//     Term 163 (AT2000-0250)/CC Inputs/Current actual value Ch.6 <-> Data Pointer/CurrentActualValues[5]
//     Term 163 (AT2000-0250)/CC Inputs/Current actual value Ch.7 <-> Data Pointer/CurrentActualValues[6]
//     Term 163 (AT2000-0250)/CC Inputs/Current actual value Ch.8 <-> Data Pointer/CurrentActualValues[7]
//     Term 163 (AT2000-0250)/CC Inputs/Current actual value Ch.9 <-> Data Pointer/CurrentActualValues[8]
//     Term 163 (AT2000-0250)/CC Inputs/Status <-> Data Pointer/Status
//     Term 163 (AT2000-0250)/CC Outputs/Control <-> Data Pointer/Control
//     Term 163 (AT2000-0250)/CC Outputs/Current setpoint value Ch.1 <-> Data Pointer/CurrentSetpointValues[0]
//     Term 163 (AT2000-0250)/CC Outputs/Current setpoint value Ch.10 <-> Data Pointer/CurrentSetpointValues[9]
//     Term 163 (AT2000-0250)/CC Outputs/Current setpoint value Ch.11 <-> Data Pointer/CurrentSetpointValues[10]
//     Term 163 (AT2000-0250)/CC Outputs/Current setpoint value Ch.12 <-> Data Pointer/CurrentSetpointValues[11]
//     Term 163 (AT2000-0250)/CC Outputs/Current setpoint value Ch.13 <-> Data Pointer/CurrentSetpointValues[12]
//     Term 163 (AT2000-0250)/CC Outputs/Current setpoint value Ch.14 <-> Data Pointer/CurrentSetpointValues[13]
//     Term 163 (AT2000-0250)/CC Outputs/Current setpoint value Ch.15 <-> Data Pointer/CurrentSetpointValues[14]
//     Term 163 (AT2000-0250)/CC Outputs/Current setpoint value Ch.2 <-> Data Pointer/CurrentSetpointValues[1]
//     Term 163 (AT2000-0250)/CC Outputs/Current setpoint value Ch.3 <-> Data Pointer/CurrentSetpointValues[2]
//     Term 163 (AT2000-0250)/CC Outputs/Current setpoint value Ch.4 <-> Data Pointer/CurrentSetpointValues[3]
//     Term 163 (AT2000-0250)/CC Outputs/Current setpoint value Ch.5 <-> Data Pointer/CurrentSetpointValues[4]
//     Term 163 (AT2000-0250)/CC Outputs/Current setpoint value Ch.6 <-> Data Pointer/CurrentSetpointValues[5]
//     Term 163 (AT2000-0250)/CC Outputs/Current setpoint value Ch.7 <-> Data Pointer/CurrentSetpointValues[6]
//     Term 163 (AT2000-0250)/CC Outputs/Current setpoint value Ch.8 <-> Data Pointer/CurrentSetpointValues[7]
//     Term 163 (AT2000-0250)/CC Outputs/Current setpoint value Ch.9 <-> Data Pointer/CurrentSetpointValues[8]
//     Term 163 (AT2000-0250)/Term 164 (AT2000-5250)/FB Inputs/Value Channel 01 <-> Data Pointer/RawPositionValues[0]
//     Term 163 (AT2000-0250)/Term 164 (AT2000-5250)/FB Inputs/Value Channel 02 <-> Data Pointer/RawPositionValues[1]
//     Term 163 (AT2000-0250)/Term 164 (AT2000-5250)/FB Inputs/Value Channel 03 <-> Data Pointer/RawPositionValues[2]
//     Term 163 (AT2000-0250)/Term 164 (AT2000-5250)/FB Inputs/Value Channel 04 <-> Data Pointer/RawPositionValues[3]
//     Term 163 (AT2000-0250)/Term 164 (AT2000-5250)/FB Inputs/Value Channel 05 <-> Data Pointer/RawPositionValues[4]
//     Term 163 (AT2000-0250)/Term 164 (AT2000-5250)/FB Inputs/Value Channel 06 <-> Data Pointer/RawPositionValues[5]
//     Term 163 (AT2000-0250)/Term 164 (AT2000-5250)/FB Inputs/Value Channel 07 <-> Data Pointer/RawPositionValues[6]
//     Term 163 (AT2000-0250)/Term 164 (AT2000-5250)/FB Inputs/Value Channel 08 <-> Data Pointer/RawPositionValues[7]
//     Term 163 (AT2000-0250)/Term 164 (AT2000-5250)/FB Inputs/Value Channel 09 <-> Data Pointer/RawPositionValues[8]
//     Term 163 (AT2000-0250)/Term 164 (AT2000-5250)/FB Inputs/Value Channel 10 <-> Data Pointer/RawPositionValues[9]
//     Term 163 (AT2000-0250)/Term 164 (AT2000-5250)/FB Inputs/Value Channel 11 <-> Data Pointer/RawPositionValues[10]
//     Term 163 (AT2000-0250)/Term 164 (AT2000-5250)/FB Inputs/Value Channel 12 <-> Data Pointer/RawPositionValues[11]
//     Term 163 (AT2000-0250)/Term 164 (AT2000-5250)/FB Inputs/Value Channel 13 <-> Data Pointer/RawPositionValues[12]
//     Term 163 (AT2000-0250)/Term 164 (AT2000-5250)/FB Inputs/Value Channel 14 <-> Data Pointer/RawPositionValues[13]
//     Term 163 (AT2000-0250)/Term 164 (AT2000-5250)/FB Inputs/Value Channel 15 <-> Data Pointer/RawPositionValues[14]
//     Term 163 (AT2000-0250)/Term 164 (AT2000-5250)/FB Inputs/Value Channel 16 <-> Data Pointer/RawPositionValues[15]
//     Term 163 (AT2000-0250)/Term 164 (AT2000-5250)/FB Inputs/Value Channel 17 <-> Data Pointer/RawPositionValues[16]
//     Term 163 (AT2000-0250)/Term 164 (AT2000-5250)/FB Inputs/Value Channel 18 <-> Data Pointer/RawPositionValues[17]
//     Term 163 (AT2000-0250)/Term 164 (AT2000-5250)/FB Inputs/Value Channel 19 <-> Data Pointer/RawPositionValues[18]
//     Term 163 (AT2000-0250)/Term 164 (AT2000-5250)/FB Inputs/Value Channel 20 <-> Data Pointer/RawPositionValues[19]
//     Term 163 (AT2000-0250)/Term 164 (AT2000-5250)/FB Inputs/Value Channel 21 <-> Data Pointer/RawPositionValues[20]
//     Term 163 (AT2000-0250)/Term 164 (AT2000-5250)/FB Inputs/Value Channel 22 <-> Data Pointer/RawPositionValues[21]
//     Term 163 (AT2000-0250)/Term 164 (AT2000-5250)/FB Inputs/Value Channel 23 <-> Data Pointer/RawPositionValues[22]
//     Term 163 (AT2000-0250)/Term 164 (AT2000-5250)/FB Inputs/Value Channel 24 <-> Data Pointer/RawPositionValues[23]
//     Term 163 (AT2000-0250)/Term 164 (AT2000-5250)/FB Inputs/Value Channel 25 <-> Data Pointer/RawPositionValues[24]
//     Term 163 (AT2000-0250)/Term 164 (AT2000-5250)/FB Inputs/Value Channel 26 <-> Data Pointer/RawPositionValues[25]
//     Term 163 (AT2000-0250)/Term 164 (AT2000-5250)/FB Inputs/Value Channel 27 <-> Data Pointer/RawPositionValues[26]
//     Term 163 (AT2000-0250)/Term 164 (AT2000-5250)/FB Inputs/Value Channel 28 <-> Data Pointer/RawPositionValues[27]
//     Term 163 (AT2000-0250)/Term 164 (AT2000-5250)/FB Inputs/Value Channel 29 <-> Data Pointer/RawPositionValues[28]
//     Term 163 (AT2000-0250)/Term 164 (AT2000-5250)/FB Inputs/Value Channel 30 <-> Data Pointer/RawPositionValues[29]
//     Term 163 (AT2000-0250)/Term 164 (AT2000-5250)/FB Inputs/Value Channel 31 <-> Data Pointer/RawPositionValues[30]
//     Term 163 (AT2000-0250)/Term 164 (AT2000-5250)/FB Inputs/Value Channel 32 <-> Data Pointer/RawPositionValues[31]
//   (this object) <-> TcCOM Objects/XtsProcessingUnit 1/Part 1/Module 83
//     Term 165 (AT2050-0500)/CC Inputs/Current actual value Ch.1 <-> Data Pointer/CurrentActualValues[0]
//     Term 165 (AT2050-0500)/CC Inputs/Current actual value Ch.10 <-> Data Pointer/CurrentActualValues[9]
//     Term 165 (AT2050-0500)/CC Inputs/Current actual value Ch.11 <-> Data Pointer/CurrentActualValues[10]
//     Term 165 (AT2050-0500)/CC Inputs/Current actual value Ch.12 <-> Data Pointer/CurrentActualValues[11]
//     Term 165 (AT2050-0500)/CC Inputs/Current actual value Ch.13 <-> Data Pointer/CurrentActualValues[12]
//     Term 165 (AT2050-0500)/CC Inputs/Current actual value Ch.14 <-> Data Pointer/CurrentActualValues[13]
//     Term 165 (AT2050-0500)/CC Inputs/Current actual value Ch.15 <-> Data Pointer/CurrentActualValues[14]
//     Term 165 (AT2050-0500)/CC Inputs/Current actual value Ch.2 <-> Data Pointer/CurrentActualValues[1]
//     Term 165 (AT2050-0500)/CC Inputs/Current actual value Ch.3 <-> Data Pointer/CurrentActualValues[2]
//     Term 165 (AT2050-0500)/CC Inputs/Current actual value Ch.4 <-> Data Pointer/CurrentActualValues[3]
//     Term 165 (AT2050-0500)/CC Inputs/Current actual value Ch.5 <-> Data Pointer/CurrentActualValues[4]
//     Term 165 (AT2050-0500)/CC Inputs/Current actual value Ch.6 <-> Data Pointer/CurrentActualValues[5]
//     Term 165 (AT2050-0500)/CC Inputs/Current actual value Ch.7 <-> Data Pointer/CurrentActualValues[6]
//     Term 165 (AT2050-0500)/CC Inputs/Current actual value Ch.8 <-> Data Pointer/CurrentActualValues[7]
//     Term 165 (AT2050-0500)/CC Inputs/Current actual value Ch.9 <-> Data Pointer/CurrentActualValues[8]
//     Term 165 (AT2050-0500)/CC Inputs/Status <-> Data Pointer/Status
//     Term 165 (AT2050-0500)/CC Outputs/Control <-> Data Pointer/Control
//     Term 165 (AT2050-0500)/CC Outputs/Current setpoint value Ch.1 <-> Data Pointer/CurrentSetpointValues[0]
//     Term 165 (AT2050-0500)/CC Outputs/Current setpoint value Ch.10 <-> Data Pointer/CurrentSetpointValues[9]
//     Term 165 (AT2050-0500)/CC Outputs/Current setpoint value Ch.11 <-> Data Pointer/CurrentSetpointValues[10]
//     Term 165 (AT2050-0500)/CC Outputs/Current setpoint value Ch.12 <-> Data Pointer/CurrentSetpointValues[11]
//     Term 165 (AT2050-0500)/CC Outputs/Current setpoint value Ch.13 <-> Data Pointer/CurrentSetpointValues[12]
//     Term 165 (AT2050-0500)/CC Outputs/Current setpoint value Ch.14 <-> Data Pointer/CurrentSetpointValues[13]
//     Term 165 (AT2050-0500)/CC Outputs/Current setpoint value Ch.15 <-> Data Pointer/CurrentSetpointValues[14]
//     Term 165 (AT2050-0500)/CC Outputs/Current setpoint value Ch.2 <-> Data Pointer/CurrentSetpointValues[1]
//     Term 165 (AT2050-0500)/CC Outputs/Current setpoint value Ch.3 <-> Data Pointer/CurrentSetpointValues[2]
//     Term 165 (AT2050-0500)/CC Outputs/Current setpoint value Ch.4 <-> Data Pointer/CurrentSetpointValues[3]
//     Term 165 (AT2050-0500)/CC Outputs/Current setpoint value Ch.5 <-> Data Pointer/CurrentSetpointValues[4]
//     Term 165 (AT2050-0500)/CC Outputs/Current setpoint value Ch.6 <-> Data Pointer/CurrentSetpointValues[5]
//     Term 165 (AT2050-0500)/CC Outputs/Current setpoint value Ch.7 <-> Data Pointer/CurrentSetpointValues[6]
//     Term 165 (AT2050-0500)/CC Outputs/Current setpoint value Ch.8 <-> Data Pointer/CurrentSetpointValues[7]
//     Term 165 (AT2050-0500)/CC Outputs/Current setpoint value Ch.9 <-> Data Pointer/CurrentSetpointValues[8]
//     Term 165 (AT2050-0500)/Term 166 (AT2050-5500)/FB Inputs/Value Channel 01 <-> Data Pointer/RawPositionValues[0]
//     Term 165 (AT2050-0500)/Term 166 (AT2050-5500)/FB Inputs/Value Channel 02 <-> Data Pointer/RawPositionValues[1]
//     Term 165 (AT2050-0500)/Term 166 (AT2050-5500)/FB Inputs/Value Channel 03 <-> Data Pointer/RawPositionValues[2]
//     Term 165 (AT2050-0500)/Term 166 (AT2050-5500)/FB Inputs/Value Channel 04 <-> Data Pointer/RawPositionValues[3]
//     Term 165 (AT2050-0500)/Term 166 (AT2050-5500)/FB Inputs/Value Channel 05 <-> Data Pointer/RawPositionValues[4]
//     Term 165 (AT2050-0500)/Term 166 (AT2050-5500)/FB Inputs/Value Channel 06 <-> Data Pointer/RawPositionValues[5]
//     Term 165 (AT2050-0500)/Term 166 (AT2050-5500)/FB Inputs/Value Channel 07 <-> Data Pointer/RawPositionValues[6]
//     Term 165 (AT2050-0500)/Term 166 (AT2050-5500)/FB Inputs/Value Channel 08 <-> Data Pointer/RawPositionValues[7]
//     Term 165 (AT2050-0500)/Term 166 (AT2050-5500)/FB Inputs/Value Channel 09 <-> Data Pointer/RawPositionValues[8]
//     Term 165 (AT2050-0500)/Term 166 (AT2050-5500)/FB Inputs/Value Channel 10 <-> Data Pointer/RawPositionValues[9]
//     Term 165 (AT2050-0500)/Term 166 (AT2050-5500)/FB Inputs/Value Channel 11 <-> Data Pointer/RawPositionValues[10]
//     Term 165 (AT2050-0500)/Term 166 (AT2050-5500)/FB Inputs/Value Channel 12 <-> Data Pointer/RawPositionValues[11]
//     Term 165 (AT2050-0500)/Term 166 (AT2050-5500)/FB Inputs/Value Channel 13 <-> Data Pointer/RawPositionValues[12]
//     Term 165 (AT2050-0500)/Term 166 (AT2050-5500)/FB Inputs/Value Channel 14 <-> Data Pointer/RawPositionValues[13]
//     Term 165 (AT2050-0500)/Term 166 (AT2050-5500)/FB Inputs/Value Channel 15 <-> Data Pointer/RawPositionValues[14]
//     Term 165 (AT2050-0500)/Term 166 (AT2050-5500)/FB Inputs/Value Channel 16 <-> Data Pointer/RawPositionValues[15]
//     Term 165 (AT2050-0500)/Term 166 (AT2050-5500)/FB Inputs/Value Channel 17 <-> Data Pointer/RawPositionValues[16]
//     Term 165 (AT2050-0500)/Term 166 (AT2050-5500)/FB Inputs/Value Channel 18 <-> Data Pointer/RawPositionValues[17]
//     Term 165 (AT2050-0500)/Term 166 (AT2050-5500)/FB Inputs/Value Channel 19 <-> Data Pointer/RawPositionValues[18]
//     Term 165 (AT2050-0500)/Term 166 (AT2050-5500)/FB Inputs/Value Channel 20 <-> Data Pointer/RawPositionValues[19]
//     Term 165 (AT2050-0500)/Term 166 (AT2050-5500)/FB Inputs/Value Channel 21 <-> Data Pointer/RawPositionValues[20]
//     Term 165 (AT2050-0500)/Term 166 (AT2050-5500)/FB Inputs/Value Channel 22 <-> Data Pointer/RawPositionValues[21]
//     Term 165 (AT2050-0500)/Term 166 (AT2050-5500)/FB Inputs/Value Channel 23 <-> Data Pointer/RawPositionValues[22]
//     Term 165 (AT2050-0500)/Term 166 (AT2050-5500)/FB Inputs/Value Channel 24 <-> Data Pointer/RawPositionValues[23]
//     Term 165 (AT2050-0500)/Term 166 (AT2050-5500)/FB Inputs/Value Channel 25 <-> Data Pointer/RawPositionValues[24]
//     Term 165 (AT2050-0500)/Term 166 (AT2050-5500)/FB Inputs/Value Channel 26 <-> Data Pointer/RawPositionValues[25]
//     Term 165 (AT2050-0500)/Term 166 (AT2050-5500)/FB Inputs/Value Channel 27 <-> Data Pointer/RawPositionValues[26]
//     Term 165 (AT2050-0500)/Term 166 (AT2050-5500)/FB Inputs/Value Channel 28 <-> Data Pointer/RawPositionValues[27]
//     Term 165 (AT2050-0500)/Term 166 (AT2050-5500)/FB Inputs/Value Channel 29 <-> Data Pointer/RawPositionValues[28]
//     Term 165 (AT2050-0500)/Term 166 (AT2050-5500)/FB Inputs/Value Channel 30 <-> Data Pointer/RawPositionValues[29]
//     Term 165 (AT2050-0500)/Term 166 (AT2050-5500)/FB Inputs/Value Channel 31 <-> Data Pointer/RawPositionValues[30]
//     Term 165 (AT2050-0500)/Term 166 (AT2050-5500)/FB Inputs/Value Channel 32 <-> Data Pointer/RawPositionValues[31]
//   (this object) <-> TcCOM Objects/XtsProcessingUnit 1/Part 1/Module 84
//     Term 167 (AT2050-0501)/CC Inputs/Current actual value Ch.1 <-> Data Pointer/CurrentActualValues[0]
//     Term 167 (AT2050-0501)/CC Inputs/Current actual value Ch.10 <-> Data Pointer/CurrentActualValues[9]
//     Term 167 (AT2050-0501)/CC Inputs/Current actual value Ch.11 <-> Data Pointer/CurrentActualValues[10]
//     Term 167 (AT2050-0501)/CC Inputs/Current actual value Ch.12 <-> Data Pointer/CurrentActualValues[11]
//     Term 167 (AT2050-0501)/CC Inputs/Current actual value Ch.13 <-> Data Pointer/CurrentActualValues[12]
//     Term 167 (AT2050-0501)/CC Inputs/Current actual value Ch.14 <-> Data Pointer/CurrentActualValues[13]
//     Term 167 (AT2050-0501)/CC Inputs/Current actual value Ch.15 <-> Data Pointer/CurrentActualValues[14]
//     Term 167 (AT2050-0501)/CC Inputs/Current actual value Ch.2 <-> Data Pointer/CurrentActualValues[1]
//     Term 167 (AT2050-0501)/CC Inputs/Current actual value Ch.3 <-> Data Pointer/CurrentActualValues[2]
//     Term 167 (AT2050-0501)/CC Inputs/Current actual value Ch.4 <-> Data Pointer/CurrentActualValues[3]
//     Term 167 (AT2050-0501)/CC Inputs/Current actual value Ch.5 <-> Data Pointer/CurrentActualValues[4]
//     Term 167 (AT2050-0501)/CC Inputs/Current actual value Ch.6 <-> Data Pointer/CurrentActualValues[5]
//     Term 167 (AT2050-0501)/CC Inputs/Current actual value Ch.7 <-> Data Pointer/CurrentActualValues[6]
//     Term 167 (AT2050-0501)/CC Inputs/Current actual value Ch.8 <-> Data Pointer/CurrentActualValues[7]
//     Term 167 (AT2050-0501)/CC Inputs/Current actual value Ch.9 <-> Data Pointer/CurrentActualValues[8]
//     Term 167 (AT2050-0501)/CC Inputs/Status <-> Data Pointer/Status
//     Term 167 (AT2050-0501)/CC Outputs/Control <-> Data Pointer/Control
//     Term 167 (AT2050-0501)/CC Outputs/Current setpoint value Ch.1 <-> Data Pointer/CurrentSetpointValues[0]
//     Term 167 (AT2050-0501)/CC Outputs/Current setpoint value Ch.10 <-> Data Pointer/CurrentSetpointValues[9]
//     Term 167 (AT2050-0501)/CC Outputs/Current setpoint value Ch.11 <-> Data Pointer/CurrentSetpointValues[10]
//     Term 167 (AT2050-0501)/CC Outputs/Current setpoint value Ch.12 <-> Data Pointer/CurrentSetpointValues[11]
//     Term 167 (AT2050-0501)/CC Outputs/Current setpoint value Ch.13 <-> Data Pointer/CurrentSetpointValues[12]
//     Term 167 (AT2050-0501)/CC Outputs/Current setpoint value Ch.14 <-> Data Pointer/CurrentSetpointValues[13]
//     Term 167 (AT2050-0501)/CC Outputs/Current setpoint value Ch.15 <-> Data Pointer/CurrentSetpointValues[14]
//     Term 167 (AT2050-0501)/CC Outputs/Current setpoint value Ch.2 <-> Data Pointer/CurrentSetpointValues[1]
//     Term 167 (AT2050-0501)/CC Outputs/Current setpoint value Ch.3 <-> Data Pointer/CurrentSetpointValues[2]
//     Term 167 (AT2050-0501)/CC Outputs/Current setpoint value Ch.4 <-> Data Pointer/CurrentSetpointValues[3]
//     Term 167 (AT2050-0501)/CC Outputs/Current setpoint value Ch.5 <-> Data Pointer/CurrentSetpointValues[4]
//     Term 167 (AT2050-0501)/CC Outputs/Current setpoint value Ch.6 <-> Data Pointer/CurrentSetpointValues[5]
//     Term 167 (AT2050-0501)/CC Outputs/Current setpoint value Ch.7 <-> Data Pointer/CurrentSetpointValues[6]
//     Term 167 (AT2050-0501)/CC Outputs/Current setpoint value Ch.8 <-> Data Pointer/CurrentSetpointValues[7]
//     Term 167 (AT2050-0501)/CC Outputs/Current setpoint value Ch.9 <-> Data Pointer/CurrentSetpointValues[8]
//     Term 167 (AT2050-0501)/Term 168 (AT2050-5501)/FB Inputs/Value Channel 01 <-> Data Pointer/RawPositionValues[0]
//     Term 167 (AT2050-0501)/Term 168 (AT2050-5501)/FB Inputs/Value Channel 02 <-> Data Pointer/RawPositionValues[1]
//     Term 167 (AT2050-0501)/Term 168 (AT2050-5501)/FB Inputs/Value Channel 03 <-> Data Pointer/RawPositionValues[2]
//     Term 167 (AT2050-0501)/Term 168 (AT2050-5501)/FB Inputs/Value Channel 04 <-> Data Pointer/RawPositionValues[3]
//     Term 167 (AT2050-0501)/Term 168 (AT2050-5501)/FB Inputs/Value Channel 05 <-> Data Pointer/RawPositionValues[4]
//     Term 167 (AT2050-0501)/Term 168 (AT2050-5501)/FB Inputs/Value Channel 06 <-> Data Pointer/RawPositionValues[5]
//     Term 167 (AT2050-0501)/Term 168 (AT2050-5501)/FB Inputs/Value Channel 07 <-> Data Pointer/RawPositionValues[6]
//     Term 167 (AT2050-0501)/Term 168 (AT2050-5501)/FB Inputs/Value Channel 08 <-> Data Pointer/RawPositionValues[7]
//     Term 167 (AT2050-0501)/Term 168 (AT2050-5501)/FB Inputs/Value Channel 09 <-> Data Pointer/RawPositionValues[8]
//     Term 167 (AT2050-0501)/Term 168 (AT2050-5501)/FB Inputs/Value Channel 10 <-> Data Pointer/RawPositionValues[9]
//     Term 167 (AT2050-0501)/Term 168 (AT2050-5501)/FB Inputs/Value Channel 11 <-> Data Pointer/RawPositionValues[10]
//     Term 167 (AT2050-0501)/Term 168 (AT2050-5501)/FB Inputs/Value Channel 12 <-> Data Pointer/RawPositionValues[11]
//     Term 167 (AT2050-0501)/Term 168 (AT2050-5501)/FB Inputs/Value Channel 13 <-> Data Pointer/RawPositionValues[12]
//     Term 167 (AT2050-0501)/Term 168 (AT2050-5501)/FB Inputs/Value Channel 14 <-> Data Pointer/RawPositionValues[13]
//     Term 167 (AT2050-0501)/Term 168 (AT2050-5501)/FB Inputs/Value Channel 15 <-> Data Pointer/RawPositionValues[14]
//     Term 167 (AT2050-0501)/Term 168 (AT2050-5501)/FB Inputs/Value Channel 16 <-> Data Pointer/RawPositionValues[15]
//     Term 167 (AT2050-0501)/Term 168 (AT2050-5501)/FB Inputs/Value Channel 17 <-> Data Pointer/RawPositionValues[16]
//     Term 167 (AT2050-0501)/Term 168 (AT2050-5501)/FB Inputs/Value Channel 18 <-> Data Pointer/RawPositionValues[17]
//     Term 167 (AT2050-0501)/Term 168 (AT2050-5501)/FB Inputs/Value Channel 19 <-> Data Pointer/RawPositionValues[18]
//     Term 167 (AT2050-0501)/Term 168 (AT2050-5501)/FB Inputs/Value Channel 20 <-> Data Pointer/RawPositionValues[19]
//     Term 167 (AT2050-0501)/Term 168 (AT2050-5501)/FB Inputs/Value Channel 21 <-> Data Pointer/RawPositionValues[20]
//     Term 167 (AT2050-0501)/Term 168 (AT2050-5501)/FB Inputs/Value Channel 22 <-> Data Pointer/RawPositionValues[21]
//     Term 167 (AT2050-0501)/Term 168 (AT2050-5501)/FB Inputs/Value Channel 23 <-> Data Pointer/RawPositionValues[22]
//     Term 167 (AT2050-0501)/Term 168 (AT2050-5501)/FB Inputs/Value Channel 24 <-> Data Pointer/RawPositionValues[23]
//     Term 167 (AT2050-0501)/Term 168 (AT2050-5501)/FB Inputs/Value Channel 25 <-> Data Pointer/RawPositionValues[24]
//     Term 167 (AT2050-0501)/Term 168 (AT2050-5501)/FB Inputs/Value Channel 26 <-> Data Pointer/RawPositionValues[25]
//     Term 167 (AT2050-0501)/Term 168 (AT2050-5501)/FB Inputs/Value Channel 27 <-> Data Pointer/RawPositionValues[26]
//     Term 167 (AT2050-0501)/Term 168 (AT2050-5501)/FB Inputs/Value Channel 28 <-> Data Pointer/RawPositionValues[27]
//     Term 167 (AT2050-0501)/Term 168 (AT2050-5501)/FB Inputs/Value Channel 29 <-> Data Pointer/RawPositionValues[28]
//     Term 167 (AT2050-0501)/Term 168 (AT2050-5501)/FB Inputs/Value Channel 30 <-> Data Pointer/RawPositionValues[29]
//     Term 167 (AT2050-0501)/Term 168 (AT2050-5501)/FB Inputs/Value Channel 31 <-> Data Pointer/RawPositionValues[30]
//     Term 167 (AT2050-0501)/Term 168 (AT2050-5501)/FB Inputs/Value Channel 32 <-> Data Pointer/RawPositionValues[31]
//   PLC1 Instance <-> NC-Task SAF/Axes/Mover Axis 1
//     PlcTask Inputs/MAIN.aMovers[1].Axis.Axis.NcToPlc <-> Outputs/ToPlc
//     PlcTask Outputs/MAIN.aMovers[1].Axis.Axis.PlcToNc <-> Inputs/FromPlc
//   PLC1 Instance <-> NC-Task SAF/Axes/Mover Axis 10
//     PlcTask Inputs/MAIN.aMovers[10].Axis.Axis.NcToPlc <-> Outputs/ToPlc
//     PlcTask Outputs/MAIN.aMovers[10].Axis.Axis.PlcToNc <-> Inputs/FromPlc
//   PLC1 Instance <-> NC-Task SAF/Axes/Mover Axis 100
//     PlcTask Inputs/MAIN.aMovers[100].Axis.Axis.NcToPlc <-> Outputs/ToPlc
//     PlcTask Outputs/MAIN.aMovers[100].Axis.Axis.PlcToNc <-> Inputs/FromPlc
//   PLC1 Instance <-> NC-Task SAF/Axes/Mover Axis 11
//     PlcTask Inputs/MAIN.aMovers[11].Axis.Axis.NcToPlc <-> Outputs/ToPlc
//     PlcTask Outputs/MAIN.aMovers[11].Axis.Axis.PlcToNc <-> Inputs/FromPlc
//   PLC1 Instance <-> NC-Task SAF/Axes/Mover Axis 12
//     PlcTask Inputs/MAIN.aMovers[12].Axis.Axis.NcToPlc <-> Outputs/ToPlc
//     PlcTask Outputs/MAIN.aMovers[12].Axis.Axis.PlcToNc <-> Inputs/FromPlc
//   PLC1 Instance <-> NC-Task SAF/Axes/Mover Axis 13
//     PlcTask Inputs/MAIN.aMovers[13].Axis.Axis.NcToPlc <-> Outputs/ToPlc
//     PlcTask Outputs/MAIN.aMovers[13].Axis.Axis.PlcToNc <-> Inputs/FromPlc
//   PLC1 Instance <-> NC-Task SAF/Axes/Mover Axis 14
//     PlcTask Inputs/MAIN.aMovers[14].Axis.Axis.NcToPlc <-> Outputs/ToPlc
//     PlcTask Outputs/MAIN.aMovers[14].Axis.Axis.PlcToNc <-> Inputs/FromPlc
//   PLC1 Instance <-> NC-Task SAF/Axes/Mover Axis 15
//     PlcTask Inputs/MAIN.aMovers[15].Axis.Axis.NcToPlc <-> Outputs/ToPlc
//     PlcTask Outputs/MAIN.aMovers[15].Axis.Axis.PlcToNc <-> Inputs/FromPlc
//   PLC1 Instance <-> NC-Task SAF/Axes/Mover Axis 16
//     PlcTask Inputs/MAIN.aMovers[16].Axis.Axis.NcToPlc <-> Outputs/ToPlc
//     PlcTask Outputs/MAIN.aMovers[16].Axis.Axis.PlcToNc <-> Inputs/FromPlc
//   PLC1 Instance <-> NC-Task SAF/Axes/Mover Axis 17
//     PlcTask Inputs/MAIN.aMovers[17].Axis.Axis.NcToPlc <-> Outputs/ToPlc
//     PlcTask Outputs/MAIN.aMovers[17].Axis.Axis.PlcToNc <-> Inputs/FromPlc
//   PLC1 Instance <-> NC-Task SAF/Axes/Mover Axis 18
//     PlcTask Inputs/MAIN.aMovers[18].Axis.Axis.NcToPlc <-> Outputs/ToPlc
//     PlcTask Outputs/MAIN.aMovers[18].Axis.Axis.PlcToNc <-> Inputs/FromPlc
//   PLC1 Instance <-> NC-Task SAF/Axes/Mover Axis 19
//     PlcTask Inputs/MAIN.aMovers[19].Axis.Axis.NcToPlc <-> Outputs/ToPlc
//     PlcTask Outputs/MAIN.aMovers[19].Axis.Axis.PlcToNc <-> Inputs/FromPlc
//   PLC1 Instance <-> NC-Task SAF/Axes/Mover Axis 2
//     PlcTask Inputs/MAIN.aMovers[2].Axis.Axis.NcToPlc <-> Outputs/ToPlc
//     PlcTask Outputs/MAIN.aMovers[2].Axis.Axis.PlcToNc <-> Inputs/FromPlc
//   PLC1 Instance <-> NC-Task SAF/Axes/Mover Axis 20
//     PlcTask Inputs/MAIN.aMovers[20].Axis.Axis.NcToPlc <-> Outputs/ToPlc
//     PlcTask Outputs/MAIN.aMovers[20].Axis.Axis.PlcToNc <-> Inputs/FromPlc
//   PLC1 Instance <-> NC-Task SAF/Axes/Mover Axis 21
//     PlcTask Inputs/MAIN.aMovers[21].Axis.Axis.NcToPlc <-> Outputs/ToPlc
//     PlcTask Outputs/MAIN.aMovers[21].Axis.Axis.PlcToNc <-> Inputs/FromPlc
//   PLC1 Instance <-> NC-Task SAF/Axes/Mover Axis 22
//     PlcTask Inputs/MAIN.aMovers[22].Axis.Axis.NcToPlc <-> Outputs/ToPlc
//     PlcTask Outputs/MAIN.aMovers[22].Axis.Axis.PlcToNc <-> Inputs/FromPlc
//   PLC1 Instance <-> NC-Task SAF/Axes/Mover Axis 23
//     PlcTask Inputs/MAIN.aMovers[23].Axis.Axis.NcToPlc <-> Outputs/ToPlc
//     PlcTask Outputs/MAIN.aMovers[23].Axis.Axis.PlcToNc <-> Inputs/FromPlc
//   PLC1 Instance <-> NC-Task SAF/Axes/Mover Axis 24
//     PlcTask Inputs/MAIN.aMovers[24].Axis.Axis.NcToPlc <-> Outputs/ToPlc
//     PlcTask Outputs/MAIN.aMovers[24].Axis.Axis.PlcToNc <-> Inputs/FromPlc
//   PLC1 Instance <-> NC-Task SAF/Axes/Mover Axis 25
//     PlcTask Inputs/MAIN.aMovers[25].Axis.Axis.NcToPlc <-> Outputs/ToPlc
//     PlcTask Outputs/MAIN.aMovers[25].Axis.Axis.PlcToNc <-> Inputs/FromPlc
//   PLC1 Instance <-> NC-Task SAF/Axes/Mover Axis 26
//     PlcTask Inputs/MAIN.aMovers[26].Axis.Axis.NcToPlc <-> Outputs/ToPlc
//     PlcTask Outputs/MAIN.aMovers[26].Axis.Axis.PlcToNc <-> Inputs/FromPlc
//   PLC1 Instance <-> NC-Task SAF/Axes/Mover Axis 27
//     PlcTask Inputs/MAIN.aMovers[27].Axis.Axis.NcToPlc <-> Outputs/ToPlc
//     PlcTask Outputs/MAIN.aMovers[27].Axis.Axis.PlcToNc <-> Inputs/FromPlc
//   PLC1 Instance <-> NC-Task SAF/Axes/Mover Axis 28
//     PlcTask Inputs/MAIN.aMovers[28].Axis.Axis.NcToPlc <-> Outputs/ToPlc
//     PlcTask Outputs/MAIN.aMovers[28].Axis.Axis.PlcToNc <-> Inputs/FromPlc
//   PLC1 Instance <-> NC-Task SAF/Axes/Mover Axis 29
//     PlcTask Inputs/MAIN.aMovers[29].Axis.Axis.NcToPlc <-> Outputs/ToPlc
//     PlcTask Outputs/MAIN.aMovers[29].Axis.Axis.PlcToNc <-> Inputs/FromPlc
//   PLC1 Instance <-> NC-Task SAF/Axes/Mover Axis 3
//     PlcTask Inputs/MAIN.aMovers[3].Axis.Axis.NcToPlc <-> Outputs/ToPlc
//     PlcTask Outputs/MAIN.aMovers[3].Axis.Axis.PlcToNc <-> Inputs/FromPlc
//   PLC1 Instance <-> NC-Task SAF/Axes/Mover Axis 30
//     PlcTask Inputs/MAIN.aMovers[30].Axis.Axis.NcToPlc <-> Outputs/ToPlc
//     PlcTask Outputs/MAIN.aMovers[30].Axis.Axis.PlcToNc <-> Inputs/FromPlc
//   PLC1 Instance <-> NC-Task SAF/Axes/Mover Axis 31
//     PlcTask Inputs/MAIN.aMovers[31].Axis.Axis.NcToPlc <-> Outputs/ToPlc
//     PlcTask Outputs/MAIN.aMovers[31].Axis.Axis.PlcToNc <-> Inputs/FromPlc
//   PLC1 Instance <-> NC-Task SAF/Axes/Mover Axis 32
//     PlcTask Inputs/MAIN.aMovers[32].Axis.Axis.NcToPlc <-> Outputs/ToPlc
//     PlcTask Outputs/MAIN.aMovers[32].Axis.Axis.PlcToNc <-> Inputs/FromPlc
//   PLC1 Instance <-> NC-Task SAF/Axes/Mover Axis 33
//     PlcTask Inputs/MAIN.aMovers[33].Axis.Axis.NcToPlc <-> Outputs/ToPlc
//     PlcTask Outputs/MAIN.aMovers[33].Axis.Axis.PlcToNc <-> Inputs/FromPlc
//   PLC1 Instance <-> NC-Task SAF/Axes/Mover Axis 34
//     PlcTask Inputs/MAIN.aMovers[34].Axis.Axis.NcToPlc <-> Outputs/ToPlc
//     PlcTask Outputs/MAIN.aMovers[34].Axis.Axis.PlcToNc <-> Inputs/FromPlc
//   PLC1 Instance <-> NC-Task SAF/Axes/Mover Axis 35
//     PlcTask Inputs/MAIN.aMovers[35].Axis.Axis.NcToPlc <-> Outputs/ToPlc
//     PlcTask Outputs/MAIN.aMovers[35].Axis.Axis.PlcToNc <-> Inputs/FromPlc
//   PLC1 Instance <-> NC-Task SAF/Axes/Mover Axis 36
//     PlcTask Inputs/MAIN.aMovers[36].Axis.Axis.NcToPlc <-> Outputs/ToPlc
//     PlcTask Outputs/MAIN.aMovers[36].Axis.Axis.PlcToNc <-> Inputs/FromPlc
//   PLC1 Instance <-> NC-Task SAF/Axes/Mover Axis 37
//     PlcTask Inputs/MAIN.aMovers[37].Axis.Axis.NcToPlc <-> Outputs/ToPlc
//     PlcTask Outputs/MAIN.aMovers[37].Axis.Axis.PlcToNc <-> Inputs/FromPlc
//   PLC1 Instance <-> NC-Task SAF/Axes/Mover Axis 38
//     PlcTask Inputs/MAIN.aMovers[38].Axis.Axis.NcToPlc <-> Outputs/ToPlc
//     PlcTask Outputs/MAIN.aMovers[38].Axis.Axis.PlcToNc <-> Inputs/FromPlc
//   PLC1 Instance <-> NC-Task SAF/Axes/Mover Axis 39
//     PlcTask Inputs/MAIN.aMovers[39].Axis.Axis.NcToPlc <-> Outputs/ToPlc
//     PlcTask Outputs/MAIN.aMovers[39].Axis.Axis.PlcToNc <-> Inputs/FromPlc
//   PLC1 Instance <-> NC-Task SAF/Axes/Mover Axis 4
//     PlcTask Inputs/MAIN.aMovers[4].Axis.Axis.NcToPlc <-> Outputs/ToPlc
//     PlcTask Outputs/MAIN.aMovers[4].Axis.Axis.PlcToNc <-> Inputs/FromPlc
//   PLC1 Instance <-> NC-Task SAF/Axes/Mover Axis 40
//     PlcTask Inputs/MAIN.aMovers[40].Axis.Axis.NcToPlc <-> Outputs/ToPlc
//     PlcTask Outputs/MAIN.aMovers[40].Axis.Axis.PlcToNc <-> Inputs/FromPlc
//   PLC1 Instance <-> NC-Task SAF/Axes/Mover Axis 41
//     PlcTask Inputs/MAIN.aMovers[41].Axis.Axis.NcToPlc <-> Outputs/ToPlc
//     PlcTask Outputs/MAIN.aMovers[41].Axis.Axis.PlcToNc <-> Inputs/FromPlc
//   PLC1 Instance <-> NC-Task SAF/Axes/Mover Axis 42
//     PlcTask Inputs/MAIN.aMovers[42].Axis.Axis.NcToPlc <-> Outputs/ToPlc
//     PlcTask Outputs/MAIN.aMovers[42].Axis.Axis.PlcToNc <-> Inputs/FromPlc
//   PLC1 Instance <-> NC-Task SAF/Axes/Mover Axis 43
//     PlcTask Inputs/MAIN.aMovers[43].Axis.Axis.NcToPlc <-> Outputs/ToPlc
//     PlcTask Outputs/MAIN.aMovers[43].Axis.Axis.PlcToNc <-> Inputs/FromPlc
//   PLC1 Instance <-> NC-Task SAF/Axes/Mover Axis 44
//     PlcTask Inputs/MAIN.aMovers[44].Axis.Axis.NcToPlc <-> Outputs/ToPlc
//     PlcTask Outputs/MAIN.aMovers[44].Axis.Axis.PlcToNc <-> Inputs/FromPlc
//   PLC1 Instance <-> NC-Task SAF/Axes/Mover Axis 45
//     PlcTask Inputs/MAIN.aMovers[45].Axis.Axis.NcToPlc <-> Outputs/ToPlc
//     PlcTask Outputs/MAIN.aMovers[45].Axis.Axis.PlcToNc <-> Inputs/FromPlc
//   PLC1 Instance <-> NC-Task SAF/Axes/Mover Axis 46
//     PlcTask Inputs/MAIN.aMovers[46].Axis.Axis.NcToPlc <-> Outputs/ToPlc
//     PlcTask Outputs/MAIN.aMovers[46].Axis.Axis.PlcToNc <-> Inputs/FromPlc
//   PLC1 Instance <-> NC-Task SAF/Axes/Mover Axis 47
//     PlcTask Inputs/MAIN.aMovers[47].Axis.Axis.NcToPlc <-> Outputs/ToPlc
//     PlcTask Outputs/MAIN.aMovers[47].Axis.Axis.PlcToNc <-> Inputs/FromPlc
//   PLC1 Instance <-> NC-Task SAF/Axes/Mover Axis 48
//     PlcTask Inputs/MAIN.aMovers[48].Axis.Axis.NcToPlc <-> Outputs/ToPlc
//     PlcTask Outputs/MAIN.aMovers[48].Axis.Axis.PlcToNc <-> Inputs/FromPlc
//   PLC1 Instance <-> NC-Task SAF/Axes/Mover Axis 49
//     PlcTask Inputs/MAIN.aMovers[49].Axis.Axis.NcToPlc <-> Outputs/ToPlc
//     PlcTask Outputs/MAIN.aMovers[49].Axis.Axis.PlcToNc <-> Inputs/FromPlc
//   PLC1 Instance <-> NC-Task SAF/Axes/Mover Axis 5
//     PlcTask Inputs/MAIN.aMovers[5].Axis.Axis.NcToPlc <-> Outputs/ToPlc
//     PlcTask Outputs/MAIN.aMovers[5].Axis.Axis.PlcToNc <-> Inputs/FromPlc
//   PLC1 Instance <-> NC-Task SAF/Axes/Mover Axis 50
//     PlcTask Inputs/MAIN.aMovers[50].Axis.Axis.NcToPlc <-> Outputs/ToPlc
//     PlcTask Outputs/MAIN.aMovers[50].Axis.Axis.PlcToNc <-> Inputs/FromPlc
//   PLC1 Instance <-> NC-Task SAF/Axes/Mover Axis 51
//     PlcTask Inputs/MAIN.aMovers[51].Axis.Axis.NcToPlc <-> Outputs/ToPlc
//     PlcTask Outputs/MAIN.aMovers[51].Axis.Axis.PlcToNc <-> Inputs/FromPlc
//   PLC1 Instance <-> NC-Task SAF/Axes/Mover Axis 52
//     PlcTask Inputs/MAIN.aMovers[52].Axis.Axis.NcToPlc <-> Outputs/ToPlc
//     PlcTask Outputs/MAIN.aMovers[52].Axis.Axis.PlcToNc <-> Inputs/FromPlc
//   PLC1 Instance <-> NC-Task SAF/Axes/Mover Axis 53
//     PlcTask Inputs/MAIN.aMovers[53].Axis.Axis.NcToPlc <-> Outputs/ToPlc
//     PlcTask Outputs/MAIN.aMovers[53].Axis.Axis.PlcToNc <-> Inputs/FromPlc
//   PLC1 Instance <-> NC-Task SAF/Axes/Mover Axis 54
//     PlcTask Inputs/MAIN.aMovers[54].Axis.Axis.NcToPlc <-> Outputs/ToPlc
//     PlcTask Outputs/MAIN.aMovers[54].Axis.Axis.PlcToNc <-> Inputs/FromPlc
//   PLC1 Instance <-> NC-Task SAF/Axes/Mover Axis 55
//     PlcTask Inputs/MAIN.aMovers[55].Axis.Axis.NcToPlc <-> Outputs/ToPlc
//     PlcTask Outputs/MAIN.aMovers[55].Axis.Axis.PlcToNc <-> Inputs/FromPlc
//   PLC1 Instance <-> NC-Task SAF/Axes/Mover Axis 56
//     PlcTask Inputs/MAIN.aMovers[56].Axis.Axis.NcToPlc <-> Outputs/ToPlc
//     PlcTask Outputs/MAIN.aMovers[56].Axis.Axis.PlcToNc <-> Inputs/FromPlc
//   PLC1 Instance <-> NC-Task SAF/Axes/Mover Axis 57
//     PlcTask Inputs/MAIN.aMovers[57].Axis.Axis.NcToPlc <-> Outputs/ToPlc
//     PlcTask Outputs/MAIN.aMovers[57].Axis.Axis.PlcToNc <-> Inputs/FromPlc
//   PLC1 Instance <-> NC-Task SAF/Axes/Mover Axis 58
//     PlcTask Inputs/MAIN.aMovers[58].Axis.Axis.NcToPlc <-> Outputs/ToPlc
//     PlcTask Outputs/MAIN.aMovers[58].Axis.Axis.PlcToNc <-> Inputs/FromPlc
//   PLC1 Instance <-> NC-Task SAF/Axes/Mover Axis 59
//     PlcTask Inputs/MAIN.aMovers[59].Axis.Axis.NcToPlc <-> Outputs/ToPlc
//     PlcTask Outputs/MAIN.aMovers[59].Axis.Axis.PlcToNc <-> Inputs/FromPlc
//   PLC1 Instance <-> NC-Task SAF/Axes/Mover Axis 6
//     PlcTask Inputs/MAIN.aMovers[6].Axis.Axis.NcToPlc <-> Outputs/ToPlc
//     PlcTask Outputs/MAIN.aMovers[6].Axis.Axis.PlcToNc <-> Inputs/FromPlc
//   PLC1 Instance <-> NC-Task SAF/Axes/Mover Axis 60
//     PlcTask Inputs/MAIN.aMovers[60].Axis.Axis.NcToPlc <-> Outputs/ToPlc
//     PlcTask Outputs/MAIN.aMovers[60].Axis.Axis.PlcToNc <-> Inputs/FromPlc
//   PLC1 Instance <-> NC-Task SAF/Axes/Mover Axis 61
//     PlcTask Inputs/MAIN.aMovers[61].Axis.Axis.NcToPlc <-> Outputs/ToPlc
//     PlcTask Outputs/MAIN.aMovers[61].Axis.Axis.PlcToNc <-> Inputs/FromPlc
//   PLC1 Instance <-> NC-Task SAF/Axes/Mover Axis 62
//     PlcTask Inputs/MAIN.aMovers[62].Axis.Axis.NcToPlc <-> Outputs/ToPlc
//     PlcTask Outputs/MAIN.aMovers[62].Axis.Axis.PlcToNc <-> Inputs/FromPlc
//   PLC1 Instance <-> NC-Task SAF/Axes/Mover Axis 63
//     PlcTask Inputs/MAIN.aMovers[63].Axis.Axis.NcToPlc <-> Outputs/ToPlc
//     PlcTask Outputs/MAIN.aMovers[63].Axis.Axis.PlcToNc <-> Inputs/FromPlc
//   PLC1 Instance <-> NC-Task SAF/Axes/Mover Axis 64
//     PlcTask Inputs/MAIN.aMovers[64].Axis.Axis.NcToPlc <-> Outputs/ToPlc
//     PlcTask Outputs/MAIN.aMovers[64].Axis.Axis.PlcToNc <-> Inputs/FromPlc
//   PLC1 Instance <-> NC-Task SAF/Axes/Mover Axis 65
//     PlcTask Inputs/MAIN.aMovers[65].Axis.Axis.NcToPlc <-> Outputs/ToPlc
//     PlcTask Outputs/MAIN.aMovers[65].Axis.Axis.PlcToNc <-> Inputs/FromPlc
//   PLC1 Instance <-> NC-Task SAF/Axes/Mover Axis 66
//     PlcTask Inputs/MAIN.aMovers[66].Axis.Axis.NcToPlc <-> Outputs/ToPlc
//     PlcTask Outputs/MAIN.aMovers[66].Axis.Axis.PlcToNc <-> Inputs/FromPlc
//   PLC1 Instance <-> NC-Task SAF/Axes/Mover Axis 67
//     PlcTask Inputs/MAIN.aMovers[67].Axis.Axis.NcToPlc <-> Outputs/ToPlc
//     PlcTask Outputs/MAIN.aMovers[67].Axis.Axis.PlcToNc <-> Inputs/FromPlc
//   PLC1 Instance <-> NC-Task SAF/Axes/Mover Axis 68
//     PlcTask Inputs/MAIN.aMovers[68].Axis.Axis.NcToPlc <-> Outputs/ToPlc
//     PlcTask Outputs/MAIN.aMovers[68].Axis.Axis.PlcToNc <-> Inputs/FromPlc
//   PLC1 Instance <-> NC-Task SAF/Axes/Mover Axis 69
//     PlcTask Inputs/MAIN.aMovers[69].Axis.Axis.NcToPlc <-> Outputs/ToPlc
//     PlcTask Outputs/MAIN.aMovers[69].Axis.Axis.PlcToNc <-> Inputs/FromPlc
//   PLC1 Instance <-> NC-Task SAF/Axes/Mover Axis 7
//     PlcTask Inputs/MAIN.aMovers[7].Axis.Axis.NcToPlc <-> Outputs/ToPlc
//     PlcTask Outputs/MAIN.aMovers[7].Axis.Axis.PlcToNc <-> Inputs/FromPlc
//   PLC1 Instance <-> NC-Task SAF/Axes/Mover Axis 70
//     PlcTask Inputs/MAIN.aMovers[70].Axis.Axis.NcToPlc <-> Outputs/ToPlc
//     PlcTask Outputs/MAIN.aMovers[70].Axis.Axis.PlcToNc <-> Inputs/FromPlc
//   PLC1 Instance <-> NC-Task SAF/Axes/Mover Axis 71
//     PlcTask Inputs/MAIN.aMovers[71].Axis.Axis.NcToPlc <-> Outputs/ToPlc
//     PlcTask Outputs/MAIN.aMovers[71].Axis.Axis.PlcToNc <-> Inputs/FromPlc
//   PLC1 Instance <-> NC-Task SAF/Axes/Mover Axis 72
//     PlcTask Inputs/MAIN.aMovers[72].Axis.Axis.NcToPlc <-> Outputs/ToPlc
//     PlcTask Outputs/MAIN.aMovers[72].Axis.Axis.PlcToNc <-> Inputs/FromPlc
//   PLC1 Instance <-> NC-Task SAF/Axes/Mover Axis 73
//     PlcTask Inputs/MAIN.aMovers[73].Axis.Axis.NcToPlc <-> Outputs/ToPlc
//     PlcTask Outputs/MAIN.aMovers[73].Axis.Axis.PlcToNc <-> Inputs/FromPlc
//   PLC1 Instance <-> NC-Task SAF/Axes/Mover Axis 74
//     PlcTask Inputs/MAIN.aMovers[74].Axis.Axis.NcToPlc <-> Outputs/ToPlc
//     PlcTask Outputs/MAIN.aMovers[74].Axis.Axis.PlcToNc <-> Inputs/FromPlc
//   PLC1 Instance <-> NC-Task SAF/Axes/Mover Axis 75
//     PlcTask Inputs/MAIN.aMovers[75].Axis.Axis.NcToPlc <-> Outputs/ToPlc
//     PlcTask Outputs/MAIN.aMovers[75].Axis.Axis.PlcToNc <-> Inputs/FromPlc
//   PLC1 Instance <-> NC-Task SAF/Axes/Mover Axis 76
//     PlcTask Inputs/MAIN.aMovers[76].Axis.Axis.NcToPlc <-> Outputs/ToPlc
//     PlcTask Outputs/MAIN.aMovers[76].Axis.Axis.PlcToNc <-> Inputs/FromPlc
//   PLC1 Instance <-> NC-Task SAF/Axes/Mover Axis 77
//     PlcTask Inputs/MAIN.aMovers[77].Axis.Axis.NcToPlc <-> Outputs/ToPlc
//     PlcTask Outputs/MAIN.aMovers[77].Axis.Axis.PlcToNc <-> Inputs/FromPlc
//   PLC1 Instance <-> NC-Task SAF/Axes/Mover Axis 78
//     PlcTask Inputs/MAIN.aMovers[78].Axis.Axis.NcToPlc <-> Outputs/ToPlc
//     PlcTask Outputs/MAIN.aMovers[78].Axis.Axis.PlcToNc <-> Inputs/FromPlc
//   PLC1 Instance <-> NC-Task SAF/Axes/Mover Axis 79
//     PlcTask Inputs/MAIN.aMovers[79].Axis.Axis.NcToPlc <-> Outputs/ToPlc
//     PlcTask Outputs/MAIN.aMovers[79].Axis.Axis.PlcToNc <-> Inputs/FromPlc
//   PLC1 Instance <-> NC-Task SAF/Axes/Mover Axis 8
//     PlcTask Inputs/MAIN.aMovers[8].Axis.Axis.NcToPlc <-> Outputs/ToPlc
//     PlcTask Outputs/MAIN.aMovers[8].Axis.Axis.PlcToNc <-> Inputs/FromPlc
//   PLC1 Instance <-> NC-Task SAF/Axes/Mover Axis 80
//     PlcTask Inputs/MAIN.aMovers[80].Axis.Axis.NcToPlc <-> Outputs/ToPlc
//     PlcTask Outputs/MAIN.aMovers[80].Axis.Axis.PlcToNc <-> Inputs/FromPlc
//   PLC1 Instance <-> NC-Task SAF/Axes/Mover Axis 81
//     PlcTask Inputs/MAIN.aMovers[81].Axis.Axis.NcToPlc <-> Outputs/ToPlc
//     PlcTask Outputs/MAIN.aMovers[81].Axis.Axis.PlcToNc <-> Inputs/FromPlc
//   PLC1 Instance <-> NC-Task SAF/Axes/Mover Axis 82
//     PlcTask Inputs/MAIN.aMovers[82].Axis.Axis.NcToPlc <-> Outputs/ToPlc
//     PlcTask Outputs/MAIN.aMovers[82].Axis.Axis.PlcToNc <-> Inputs/FromPlc
//   PLC1 Instance <-> NC-Task SAF/Axes/Mover Axis 83
//     PlcTask Inputs/MAIN.aMovers[83].Axis.Axis.NcToPlc <-> Outputs/ToPlc
//     PlcTask Outputs/MAIN.aMovers[83].Axis.Axis.PlcToNc <-> Inputs/FromPlc
//   PLC1 Instance <-> NC-Task SAF/Axes/Mover Axis 84
//     PlcTask Inputs/MAIN.aMovers[84].Axis.Axis.NcToPlc <-> Outputs/ToPlc
//     PlcTask Outputs/MAIN.aMovers[84].Axis.Axis.PlcToNc <-> Inputs/FromPlc
//   PLC1 Instance <-> NC-Task SAF/Axes/Mover Axis 85
//     PlcTask Inputs/MAIN.aMovers[85].Axis.Axis.NcToPlc <-> Outputs/ToPlc
//     PlcTask Outputs/MAIN.aMovers[85].Axis.Axis.PlcToNc <-> Inputs/FromPlc
//   PLC1 Instance <-> NC-Task SAF/Axes/Mover Axis 86
//     PlcTask Inputs/MAIN.aMovers[86].Axis.Axis.NcToPlc <-> Outputs/ToPlc
//     PlcTask Outputs/MAIN.aMovers[86].Axis.Axis.PlcToNc <-> Inputs/FromPlc
//   PLC1 Instance <-> NC-Task SAF/Axes/Mover Axis 87
//     PlcTask Inputs/MAIN.aMovers[87].Axis.Axis.NcToPlc <-> Outputs/ToPlc
//     PlcTask Outputs/MAIN.aMovers[87].Axis.Axis.PlcToNc <-> Inputs/FromPlc
//   PLC1 Instance <-> NC-Task SAF/Axes/Mover Axis 88
//     PlcTask Inputs/MAIN.aMovers[88].Axis.Axis.NcToPlc <-> Outputs/ToPlc
//     PlcTask Outputs/MAIN.aMovers[88].Axis.Axis.PlcToNc <-> Inputs/FromPlc
//   PLC1 Instance <-> NC-Task SAF/Axes/Mover Axis 89
//     PlcTask Inputs/MAIN.aMovers[89].Axis.Axis.NcToPlc <-> Outputs/ToPlc
//     PlcTask Outputs/MAIN.aMovers[89].Axis.Axis.PlcToNc <-> Inputs/FromPlc
//   PLC1 Instance <-> NC-Task SAF/Axes/Mover Axis 9
//     PlcTask Inputs/MAIN.aMovers[9].Axis.Axis.NcToPlc <-> Outputs/ToPlc
//     PlcTask Outputs/MAIN.aMovers[9].Axis.Axis.PlcToNc <-> Inputs/FromPlc
//   PLC1 Instance <-> NC-Task SAF/Axes/Mover Axis 90
//     PlcTask Inputs/MAIN.aMovers[90].Axis.Axis.NcToPlc <-> Outputs/ToPlc
//     PlcTask Outputs/MAIN.aMovers[90].Axis.Axis.PlcToNc <-> Inputs/FromPlc
//   PLC1 Instance <-> NC-Task SAF/Axes/Mover Axis 91
//     PlcTask Inputs/MAIN.aMovers[91].Axis.Axis.NcToPlc <-> Outputs/ToPlc
//     PlcTask Outputs/MAIN.aMovers[91].Axis.Axis.PlcToNc <-> Inputs/FromPlc
//   PLC1 Instance <-> NC-Task SAF/Axes/Mover Axis 92
//     PlcTask Inputs/MAIN.aMovers[92].Axis.Axis.NcToPlc <-> Outputs/ToPlc
//     PlcTask Outputs/MAIN.aMovers[92].Axis.Axis.PlcToNc <-> Inputs/FromPlc
//   PLC1 Instance <-> NC-Task SAF/Axes/Mover Axis 93
//     PlcTask Inputs/MAIN.aMovers[93].Axis.Axis.NcToPlc <-> Outputs/ToPlc
//     PlcTask Outputs/MAIN.aMovers[93].Axis.Axis.PlcToNc <-> Inputs/FromPlc
//   PLC1 Instance <-> NC-Task SAF/Axes/Mover Axis 94
//     PlcTask Inputs/MAIN.aMovers[94].Axis.Axis.NcToPlc <-> Outputs/ToPlc
//     PlcTask Outputs/MAIN.aMovers[94].Axis.Axis.PlcToNc <-> Inputs/FromPlc
//   PLC1 Instance <-> NC-Task SAF/Axes/Mover Axis 95
//     PlcTask Inputs/MAIN.aMovers[95].Axis.Axis.NcToPlc <-> Outputs/ToPlc
//     PlcTask Outputs/MAIN.aMovers[95].Axis.Axis.PlcToNc <-> Inputs/FromPlc
//   PLC1 Instance <-> NC-Task SAF/Axes/Mover Axis 96
//     PlcTask Inputs/MAIN.aMovers[96].Axis.Axis.NcToPlc <-> Outputs/ToPlc
//     PlcTask Outputs/MAIN.aMovers[96].Axis.Axis.PlcToNc <-> Inputs/FromPlc
//   PLC1 Instance <-> NC-Task SAF/Axes/Mover Axis 97
//     PlcTask Inputs/MAIN.aMovers[97].Axis.Axis.NcToPlc <-> Outputs/ToPlc
//     PlcTask Outputs/MAIN.aMovers[97].Axis.Axis.PlcToNc <-> Inputs/FromPlc
//   PLC1 Instance <-> NC-Task SAF/Axes/Mover Axis 98
//     PlcTask Inputs/MAIN.aMovers[98].Axis.Axis.NcToPlc <-> Outputs/ToPlc
//     PlcTask Outputs/MAIN.aMovers[98].Axis.Axis.PlcToNc <-> Inputs/FromPlc
//   PLC1 Instance <-> NC-Task SAF/Axes/Mover Axis 99
//     PlcTask Inputs/MAIN.aMovers[99].Axis.Axis.NcToPlc <-> Outputs/ToPlc
//     PlcTask Outputs/MAIN.aMovers[99].Axis.Axis.PlcToNc <-> Inputs/FromPlc
//   PLC1 Instance <-> NC-Task SAF/Objects/Group1 (CA Group)
//     PlcTask Inputs/MAIN.fbGroup.GroupRef.NcToPlc <-> Group Outputs/ToPLC
//     PlcTask Outputs/MAIN.fbGroup.GroupRef.PlcToNc <-> Group Inputs/FromPLC

CONFIGURATION PLC1
    RESOURCE PLC ON TwinCAT3
        TASK PlcTask(INTERVAL := T#10ms, PRIORITY := 20);
        PROGRAM MAIN WITH PlcTask : MAIN;
    END_RESOURCE
END_CONFIGURATION

// ---- POUs/Example Product Data/I_ProductDataA.TcIO
INTERFACE I_ProductDataA EXTENDS I_XTS_ProductData

{attribute 'monitoring':='call'}
PROPERTY Data : REFERENCE TO ST_ProductDataA
GET
END_GET
END_PROPERTY

END_INTERFACE

// ---- POUs/MAIN.TcPOU
PROGRAM MAIN
VAR
	bInitDone,bDisable : BOOL;
	bEnable : BOOL;
	bStart : BOOL;
	bPreventMoversFromEntering: BOOL;

	nLoopIndex : UDINT;
	nIdxParentStation, nIdxTargedStation : UINT;
	bStandard, bRestart, bFast : BOOL;
	bStartSimulation, bStopSimulation : BOOL ;
	
	//Example of an external function block that contains the process step of the station.
	fbProcessStationXXX : FB_Station_XXX;
	
	//////////////////////////////////////////////////////////////////////////
	
	(* XTS System - 1 per associated XTS 
		The system is the container and organizer for all subsequent XTS objects. All objects are registered with this system*)
	fbSystem		: CHALET_Xts.FB_XTS_System;
	ipXtsSystem 	: CHALET_Xts.I_XTS_System_PLC := fbSystem;
		
	(* XTS Collision Avoidance Groupe - 1 per associated XTS 
		The CA group is a software object that prevents collisions between movers. 
		When the system is enabled, all movers are added to the group. As a result, only move commands with CA are permitted from this point onwards
		e.g. FB_MoveRelativeCA*)
	fbGroup			: CHALET_Xts.FB_XTS_Group(ipXtsSystem := fbSystem);
	
	(* XTS Environment - 1 per associated XTS 
		The XTS Envirement is a pure software object and offers an interface to the UtilityEnvirement and to important system information such as track length *)
	fbEnvironment	: CHALET_Xts.FB_XTS_Environment(ipXtsSystem := fbSystem);
	
	(* XTS mover - n per associated XTS. Can be instantiated as an array and/or individually *)
	aMovers		: ARRAY[1..cNrOfMovers] OF CHALET_Xts.FB_XTS_Mover(ipXtsSystem := fbSystem);
	
	(* XTS station - n per associated XTS. Can be instantiated as an array and/or individually
	The stations are the main component of the application. As soon as the system has been started up, the movers are only sent from one station to the next.
	Parameters:
		fPositionOnTrack	= Absolute position of the station on the track
		sUniqueName 		= Unique name that may only exist once. A STRING constant makes sense
		nMoverQueueSize 	= There is room for so many movers. 
							  Only when all the required movers are present is the ready signal given to the process above.
							  This parameter can also be written online
		fMoverGapAtExit		= This gap between the movers is active as soon as the mover leaves or crosses the station
							  This parameter can also be written online
		fMoverVelocityAtExit= This velocity of the movers is active as soon as the mover leaves or crosses the station
							  This parameter can also be written online	*)	
	aStations 	: ARRAY[1..cNrOfStations] OF CHALET_Xts.FB_XTS_Station[		
												(ipXtsSystem 		:= fbSystem,
												fPositionOnTrack	:= 800,
												sUniqueName			:= 'StationA_Waiting',
												nMoverQueueSize		:= 6,
												fMoverGapAtExit		:= 80,
												fMoverVelocityAtExit := 2000),
										
												(ipXtsSystem 		:= fbSystem,
												fPositionOnTrack	:= 1000,
												sUniqueName			:= 'StationA',
												nMoverQueueSize		:= 1,
												fMoverGapAtExit		:= 100,
												fMoverVelocityAtExit := 2000),
																							
												(ipXtsSystem 		:= fbSystem,
												fPositionOnTrack	:= 1500,
												sUniqueName			:= 'StationB_Waiting',
												nMoverQueueSize		:= 2,
												fMoverGapAtExit		:= 100,
												fMoverVelocityAtExit := 1000),
																																			
												(ipXtsSystem 		:= fbSystem,
												fPositionOnTrack	:= 2000,
												sUniqueName			:= 'StationB',
												nMoverQueueSize		:= 2,
												fMoverGapAtExit		:= 100,
												fMoverVelocityAtExit := 1000),
																								
												(ipXtsSystem 		:= fbSystem,
												fPositionOnTrack	:= 2500,
												sUniqueName			:= 'StationC_Waiting',
												nMoverQueueSize		:= 2,
												fMoverGapAtExit		:= 100,
												fMoverVelocityAtExit := 1000),
																								
												(ipXtsSystem 		:= fbSystem,
												fPositionOnTrack	:= 3000,
												sUniqueName			:= 'StationC',
												nMoverQueueSize		:= 3,
												fMoverGapAtExit		:= 60,
												fMoverVelocityAtExit := 1000),
																																			
												(ipXtsSystem 		:= fbSystem,
												fPositionOnTrack	:= 3500,
												sUniqueName			:= 'StationD_Waiting',
												nMoverQueueSize		:= 5,
												fMoverGapAtExit		:= 100,
												fMoverVelocityAtExit := 1000),
													
												(ipXtsSystem 		:= fbSystem,
												fPositionOnTrack	:= 4000,
												sUniqueName			:= 'StationD',
												nMoverQueueSize		:= 4,
												fMoverGapAtExit		:= 100,
												fMoverVelocityAtExit := 1000),
																																			
												(ipXtsSystem 		:= fbSystem,
												fPositionOnTrack	:= 4500,
												sUniqueName			:= 'StationE_Waiting',
												nMoverQueueSize		:= 5,
												fMoverGapAtExit		:= 100,
												fMoverVelocityAtExit := 1000),
													
												(ipXtsSystem 		:= fbSystem,
												fPositionOnTrack	:= 5000,
												sUniqueName			:= 'StationE',
												nMoverQueueSize		:= 2,
												fMoverGapAtExit		:= 100,
												fMoverVelocityAtExit := 1000),
																																			
												(ipXtsSystem 		:= fbSystem,
												fPositionOnTrack	:= 5500,
												sUniqueName			:= 'StationF_Waiting',
												nMoverQueueSize		:= 2,
												fMoverGapAtExit		:= 100,
												fMoverVelocityAtExit := 1000),
													
												(ipXtsSystem 		:= fbSystem,
												fPositionOnTrack	:= 6000,
												sUniqueName			:= 'StationF',
												nMoverQueueSize		:= 4,
												fMoverGapAtExit		:= 80,
												fMoverVelocityAtExit := 1000),
																																			
												(ipXtsSystem 		:= fbSystem,
												fPositionOnTrack	:= 6500,
												sUniqueName			:= 'StationG_Waiting',
												nMoverQueueSize		:= 2,
												fMoverGapAtExit		:= 100,
												fMoverVelocityAtExit := 1000),
													
												(ipXtsSystem 		:= fbSystem,
												fPositionOnTrack	:= 7000,
												sUniqueName			:= 'StationG',
												nMoverQueueSize		:= 5,
												fMoverGapAtExit		:= 100,
												fMoverVelocityAtExit := 1000),
																																		
												(ipXtsSystem 		:= fbSystem,
												fPositionOnTrack	:= 7500,
												sUniqueName			:= 'StationH_Waiting',
												nMoverQueueSize		:= 2,
												fMoverGapAtExit		:= 100,
												fMoverVelocityAtExit := 1000),
														
												(ipXtsSystem 		:= fbSystem,
												fPositionOnTrack	:= 8000,
												sUniqueName			:= 'StationH',
												nMoverQueueSize		:= 3,
												fMoverGapAtExit		:= 100,
												fMoverVelocityAtExit := 1000),
																																			
												(ipXtsSystem 		:= fbSystem,
												fPositionOnTrack	:= 8500,
												sUniqueName			:= 'StationI_Waiting',
												nMoverQueueSize		:= 5,
												fMoverGapAtExit		:= 100,
												fMoverVelocityAtExit := 2000),
													
												(ipXtsSystem 		:= fbSystem,
												fPositionOnTrack	:= 9000,
												sUniqueName			:= 'StationI',
												nMoverQueueSize		:= 1,
												fMoverGapAtExit		:= 100,
												fMoverVelocityAtExit := 2000),
																																			
												(ipXtsSystem 		:= fbSystem,
												fPositionOnTrack	:= 9500,
												sUniqueName			:= 'StationJ_Waiting',
												nMoverQueueSize		:= 2,
												fMoverGapAtExit		:= 100,
												fMoverVelocityAtExit := 1000),
													
												(ipXtsSystem 		:= fbSystem,
												fPositionOnTrack	:= 10000,
												sUniqueName			:= 'StationJ',
												nMoverQueueSize		:= 2,
												fMoverGapAtExit		:= 100,
												fMoverVelocityAtExit := 500),
													
												(ipXtsSystem 		:= fbSystem,
												fPositionOnTrack	:= 10500,
												sUniqueName			:= 'StationCurv1Out',
												nMoverQueueSize		:= 0,
												fMoverGapAtExit		:= 70,
												fMoverVelocityAtExit := 2000),
												
												(ipXtsSystem 		:= fbSystem,
												fPositionOnTrack	:= 20000,
												sUniqueName			:= 'StationZ_Waiting',
												nMoverQueueSize		:= 100,
												fMoverGapAtExit		:= 100,
												fMoverVelocityAtExit := 1500),
												
												(ipXtsSystem 		:= fbSystem,
												fPositionOnTrack	:= 20500,
												sUniqueName			:= 'StationCurv2In',
												nMoverQueueSize		:= 0,
												fMoverGapAtExit		:= 80,
												fMoverVelocityAtExit := 250),
												
												(ipXtsSystem 		:= fbSystem,
												fPositionOnTrack	:= 0,
												sUniqueName			:= 'StationCurv2Out',
												nMoverQueueSize		:= 0,
												fMoverGapAtExit		:= 100,
												fMoverVelocityAtExit := 1500)  
												];															
END_VAR
VAR CONSTANT
	cNrOfMovers : USINT := 100;
	cNrOfStations : USINT := 24;
END_VAR

/// Todo in a new Tc project:
/// - Add CA-Groupe + link to PLC (in MOTION\NC-Task-SAF\Objects)
/// - Set raillength in CA-Groupe
/// - Add XtsInfoServer in TcCOM. Add as many XtsStationInfos as required. Increase StopPositions to Array of size 25.
/// - Info Server: Stations link ObjectId in PLC1 Instance. 
/// -


// As long as the initialization is not completed, skip the rest of the program.
IF NOT bInitDone THEN
	fbSystem.Initialize();
	bInitDone := fbSystem.Initialized;
	
	//Handover interface to process station
	fbProcessStationXXX.ipXtsSystem := ipXtsSystem;
	fbProcessStationXXX.ipStation := ipXtsSystem.Station('StationI');
	RETURN;
END_IF


// "Start up": add the mover to the CA group, search Mover1, enable Groupe, enable Mover. No Movement
IF bEnable AND ipXtsSystem.Initialized AND ipXtsSystem.Disabled THEN
	bEnable := FALSE;	
	ipXtsSystem.Enable();
END_IF


// "Shutdown": Halt Mover, disable Mover, disable Groupe, reset Groupe, reset Mover, remove Mover from Groupe
IF bDisable THEN
	bDisable := FALSE;
	ipXtsSystem.Disable();
END_IF

// First Startup strategy: 
// Send all movers to the "Unload" station.
IF bStart AND ipXtsSystem.Enabled THEN
	bStart := FALSE;
	ipXtsSystem.SuppressAllDynamicsChanges := TRUE;	
	
	// Delete all Queues
	FOR nLoopIndex := 1 TO cNrOfStations DO
		aStations[nLoopIndex].DeleteMoversQueue();
	END_FOR	
	
	// Move + add all mover in parent station 1 (StationA_Waiting). Set as targed station 2 (StationA)
	//(the parent station is not necessarily the target station. But the station that is responsible for sending the mover forward if necessary)
	nIdxTargedStation  := 2;	
	nIdxParentStation := 1;
	FOR nLoopIndex := 1 TO cNrOfMovers DO
		aMovers[nLoopIndex].TargedStation := aStations[nIdxTargedStation].LUID;
		aMovers[nLoopIndex].MoveAbsCA(	fPosition	:=aStations[nIdxParentStation].PositionOnTrack, 
										fVelocity 	:= 1000, 
										fGap 		:= aStations[nIdxParentStation].StationBehinde.MoverGapAtExit, 
										eDirection 	:= Tc3_Mc3Definitions.MC_DIRECTION.mcDirectionPositive);
		aStations[nIdxParentStation].AddMoverToQueue(aMovers[nLoopIndex]);
	END_FOR
END_IF


// Restart strategy: 
// Send all movers to the last known parent station.
//(the parent station is not necessarily the target station. But the station that is responsible for sending the mover forward if necessary)
IF bRestart AND ipXtsSystem.Enabled THEN
	bRestart := FALSE;
	FOR nLoopIndex := 1 TO cNrOfMovers DO
		IF aMovers[nLoopIndex].ParentStation <> 0 THEN
			aMovers[nLoopIndex].MoveAbsCA(	fPosition	:= aMovers[nLoopIndex].ParentStation.PositionOnTrack, 
								fVelocity 	:= aMovers[nLoopIndex].LastCmdTargedVelocity,  
								fGap 		:= aMovers[nLoopIndex].LastCmdTargedGap,  
								eDirection 	:= Tc3_Mc3Definitions.MC_DIRECTION.mcDirectionPositive);
		END_IF
	END_FOR
END_IF


// Configure and Start Simulation
IF bStartSimulation THEN
	bStartSimulation := FALSE;
	ipXtsSystem.SuppressAllDynamicsChanges := FALSE;	//Enable to adjust Gap + Dynamic depending on Station
	ipXtsSystem.Station('StationA').SimulationMode(fProcessDuration := 0.5, sTargedStation := 'StationB');
	ipXtsSystem.Station('StationB').SimulationMode(fProcessDuration := 1.0, sTargedStation := 'StationC');
	ipXtsSystem.Station('StationC').SimulationMode(fProcessDuration := 1.5, sTargedStation := 'StationD');
	ipXtsSystem.Station('StationD').SimulationMode(fProcessDuration := 3.0, sTargedStation := 'StationE');
	ipXtsSystem.Station('StationE').SimulationMode(fProcessDuration := 1.0, sTargedStation := 'StationF');
	ipXtsSystem.Station('StationF').SimulationMode(fProcessDuration := 2.0, sTargedStation := 'StationG');
	ipXtsSystem.Station('StationG').SimulationMode(fProcessDuration := 2.5, sTargedStation := 'StationH');
	ipXtsSystem.Station('StationH').SimulationMode(fProcessDuration := 1.8, sTargedStation := 'StationI');
	
	//Station I: See "Example How to interact with process"
	//XtsSystem.Station('StationI').SimulationMode(fProcessDuration := 0.001, sTargedStation := 'StationJ');
	
	ipXtsSystem.Station('StationJ').SimulationMode(fProcessDuration := 1.0, sTargedStation := 'StationA');

END_IF

// Stop Simulation
IF bStopSimulation THEN
	bStopSimulation := FALSE;
	FOR nLoopIndex := 1 TO cNrOfStations DO
		aStations[nLoopIndex].SimulationMode(0,'');
	END_FOR	
END_IF

// Prevent further movers from entering the station, 
// e.g. to prevent a collision. All movers that are already moving to reach this station will be stopped with a stop 
// and restarted with Ready True.
ipXtsSystem.Station('StationA').ReadyToRecvMovers := NOT bPreventMoversFromEntering; //Toggle this 


// Changing of Gap Mode for Group (including Control Direction!)
// changes control direction to positiv and mode to fast
IF bFast AND ipXtsSystem.Disabled THEN
	bFast := FALSE;
	fbGroup.ChangeGapMode(bFast:= TRUE);
END_IF


// Changes mode to standard and control direction to both
IF bStandard AND ipXtsSystem.Disabled THEN
	bStandard := FALSE;
	fbGroup.ChangeGapMode(bFast:= FALSE);
END_IF


PRG_Example_ProductData_Simple();
//Simple or Advanced. Do not activate both
//PRG_Example_ProductData_Advanced();


//Update system at the end
fbSystem.Update();
fbProcessStationXXX.Update();

END_PROGRAM

// ---- POUs/Example How to interact with process/FB_Station_XXX.TcPOU
FUNCTION_BLOCK FB_Station_XXX
VAR_INPUT
	//Interface to XTS-Station and XTS-System
	ipStation : I_XTS_Station_PLC;
	ipXtsSystem : I_XTS_System_PLC; 
END_VAR
VAR
END_VAR

METHOD Update : HRESULT
VAR_INST
	nSeq : UINT;
	
END_VAR
VAR
	fTargedPos : LREAL;
	sLUIDStationAhead : STRING;
END_VAR
IF ipStation = 0  OR ipXtsSystem = 0 THEN
	RETURN; // ERROR
END_IF

IF ipXtsSystem.Disabled THEN
	nSeq := 0;
END_IF

CASE nSeq OF 

	0: //wait for mover
		IF ipStation.MoversInPlace THEN
			nSeq := 1;
		END_IF
		
	1: //Move backwards
		fTargedPos := ipStation.PositionOnTrack - 120.0;
		ipStation.MoversInQueue[0].FullAccess.MoveAbsCA(fPosition := fTargedPos, 
														fVelocity := 500, 
														fGap := 300, 
														eDirection := Tc3_Mc3Definitions.MC_DIRECTION.mcDirectionShortestWay);
		nSeq := 2;				

	2: // wait until move is finish
		IF ipStation.MoversInQueue[0].FullAccess.Feedback.Done THEN
			nSeq := 3;	
		END_IF
		
	3: //Move backwards
		fTargedPos := ipStation.PositionOnTrack;
		ipStation.MoversInQueue[0].FullAccess.MoveAbsCA(fPosition := fTargedPos, 
														fVelocity := 500, 
														fGap := 300, 
														eDirection := Tc3_Mc3Definitions.MC_DIRECTION.mcDirectionShortestWay);
		nSeq := 4;				

	4: // wait until move is finish
		IF ipStation.MoversInQueue[0].FullAccess.Feedback.Done THEN
			nSeq := 5;	
		END_IF
		
	5: // send movers away
		sLUIDStationAhead := 'StationJ';
		ipStation.SendMoversToStation(sLUIDStationAhead);
		nSeq := 0;	
	
END_CASE
END_METHOD

END_FUNCTION_BLOCK

// ---- POUs/Example Product Data/PRG_Example_ProductData_Simple.TcPOU
PROGRAM PRG_Example_ProductData_Simple
VAR
	bInitDone : BOOL;
		
	aProductsFormatA 		: ARRAY[1..MAIN.cNrOfMovers] OF FB_ProductDataA;

	ipMover					: I_XTS_Mover_PLC;
	ipProductDataOnMover 	: I_ProductDataA;

	ipStationModify 		: I_XTS_Station_PLC;
	fbTriggerMoverInPlace : R_TRIG; 
	
	nIdx : UDINT;
END_VAR

(* This example shows how easy it is to access the product data on the Mover. 
   The structure "ST_ProductDataA" can be edited to change the contained data.*)

//Do this once during initialization
IF NOT bInitDone THEN
	bInitDone := TRUE;
	
	//A separate FB with product data is added to each mover
	FOR nIdx := 1 TO MAIN.cNrOfMovers DO
		ipMover := MAIN.aMovers[nIdx]; 
		ipMover.ProductData := aProductsFormatA[nIdx];
	END_FOR
END_IF



//Get interface to StationB
ipStationModify := MAIN.ipXtsSystem.Station('StationB');
IF ipStationModify = 0 THEN
	//Abort on invalide interface
	RETURN;
END_IF

//This is executed once when the mover arrives at the station
fbTriggerMoverInPlace(CLK:= ipStationModify.MoversInPlace);
IF fbTriggerMoverInPlace.Q THEN
	
	//Do this for each mover inside the station
	FOR nIdx := 0 TO (ipStationModify.MoverQueueSize-1) DO
		
		//Query whether the FB behind this instance implements the following interface and get it.
		IF __QUERYINTERFACE(ipStationModify.MoversInQueue[nIdx].ProductData, ipProductDataOnMover) THEN 
			//Modify data
			ipProductDataOnMover.Data.nQuality 		:= (ipProductDataOnMover.Data.nQuality + 42)MOD 100;	
			ipProductDataOnMover.Data.bGoodProduct 	:= ipProductDataOnMover.Data.nQuality >= 80;
		END_IF
	
	END_FOR
END_IF

END_PROGRAM

// ---- POUs/Example Product Data/FB_ProductDataA.TcPOU
FUNCTION_BLOCK FB_ProductDataA EXTENDS FB_XTS_ProductData IMPLEMENTS I_ProductDataA
VAR
	{attribute 'hide'}	
	stData 	: ST_ProductDataA;
END_VAR

{attribute 'monitoring':='call'}
PROPERTY Data : REFERENCE TO ST_ProductDataA
GET
Data REF= stData;
END_GET
END_PROPERTY

END_FUNCTION_BLOCK

// ---- POUs/Example Product Data/PRG_Example_ProductData_Advanced.TcPOU
PROGRAM PRG_Example_ProductData_Advanced
VAR
	bInitDone : BOOL;
		
	aProductsFormatA 	: ARRAY[0..(MAIN.cNrOfMovers-1)] OF FB_ProductDataA;
	fbProductsUnused 	: CHALET_BaseComponents.FB_CH_List; //In this example this list is used to transfer products to the XTS
	fbProductsOnMover 	: CHALET_BaseComponents.FB_CH_List; //As long as the products are on the XTS, each of them can be reached via this list and the interface to the mover can also be requested.
	
	ipObject 			: I_CH_Object;
	ipProductFormatA 	: I_ProductDataA;

	ipStationLoad, ipStationModify, ipStationUnload : I_XTS_Station_PLC;
	fbTriggerMoverInPlace1, fbTriggerMoverInPlace2, fbTriggerMoverInPlace3 : R_TRIG; 
	
	nIdx : UDINT;
END_VAR

(* 
   This extended example shows how existing product data from a previous process is loaded onto the mover in StationA (e.g. robot). 
   This information is then processed in StationB (e.g. camera). 
   Finally, the product information is removed from the mover in StationC and transferred to the next process step outside the XTS 
*)

//Do this once during initialization
IF NOT bInitDone THEN
	bInitDone := TRUE;
	
	//Put all product informations in a list to easy access them
	FOR nIdx := 0 TO (MAIN.cNrOfMovers-1) DO
		fbProductsUnused.AddObject(aProductsFormatA[nIdx]);
	END_FOR
END_IF



//Station A: put empty product info FB on mover
ipStationLoad := MAIN.ipXtsSystem.Station('StationA');
IF ipStationLoad = 0 THEN
	//Abort on invalide interface
	RETURN;
END_IF

//This is executed once when the mover arrives at the station
fbTriggerMoverInPlace1(CLK:= ipStationLoad.MoversInPlace);
IF fbTriggerMoverInPlace1.Q THEN
	//Do this for each mover inside the station
	FOR nIdx := 0 TO (ipStationLoad.MoverQueueSize-1) DO
		
		// Only execute if datacontainer on mover is empty
		IF ipStationLoad.MoversInQueue[nIdx].ProductData = 0 THEN
			
			//Get an unused product OR handover here the product data from the previous process step here
			ipObject := fbProductsUnused.GetRandomObject();
			
			//Remove an put in OnMovers List
			fbProductsUnused.RemoveObject(ipObject);
			fbProductsOnMover.AddObject(ipObject);
			
			
			//Query whether the FB behind this instance implements the following interface and get it.
			IF __QUERYINTERFACE(ipObject, ipProductFormatA) THEN		
				//Store the interface in the Mover
				ipStationLoad.MoversInQueue[nIdx].ProductData := ipProductFormatA; // <= one of the important steps. Everything else around is application specific
			END_IF
		
		END_IF
		

	END_FOR
END_IF


//Station B: read/write product info 
ipStationModify := MAIN.ipXtsSystem.Station('StationB');
IF ipStationModify = 0 THEN
	//Abort on invalide interface
	RETURN;
END_IF
//This is executed once when the mover arrives at the station
fbTriggerMoverInPlace2(CLK:= ipStationModify.MoversInPlace);
IF fbTriggerMoverInPlace2.Q THEN
	//Do this for each mover inside the station
	FOR nIdx := 0 TO (ipStationModify.MoverQueueSize-1) DO
		
		//Query whether the FB behind this instance implements the following interface and get it.
		IF __QUERYINTERFACE(ipStationModify.MoversInQueue[nIdx].ProductData, ipProductFormatA) THEN // <= one of the important steps. Everything else around is application specific
			ipProductFormatA.Data.nQuality := (ipProductFormatA.Data.nQuality + 42)MOD 100;	
			ipProductFormatA.Data.bGoodProduct := ipProductFormatA.Data.nQuality >= 80;
		END_IF
	
	END_FOR
END_IF



//Station C: Remove Produkt from XTS
ipStationUnload := MAIN.ipXtsSystem.Station('StationC');
IF ipStationUnload = 0 THEN
	//Abort on invalide interface
	RETURN;
END_IF
//This is executed once when the mover arrives at the station
fbTriggerMoverInPlace3(CLK:= ipStationUnload.MoversInPlace);
IF fbTriggerMoverInPlace3.Q THEN
	//Do this for each mover inside the station
	FOR nIdx := 0 TO (ipStationUnload.MoverQueueSize-1) DO
		
		//Query whether the FB behind this instance implements the following interface and get it.
		IF __QUERYINTERFACE(ipStationUnload.MoversInQueue[nIdx].ProductData, ipObject) THEN
			
			//Handover to next processing unit OR in this case, put in UnusedList
			fbProductsOnMover.RemoveObject(ipObject);
			fbProductsUnused.AddObject(ipObject);
		END_IF
		
		// Clear mover storage
		ipStationUnload.MoversInQueue[nIdx].ProductData := 0; // <= one of the important steps. Everything else around is application specific
	END_FOR
END_IF

END_PROGRAM
